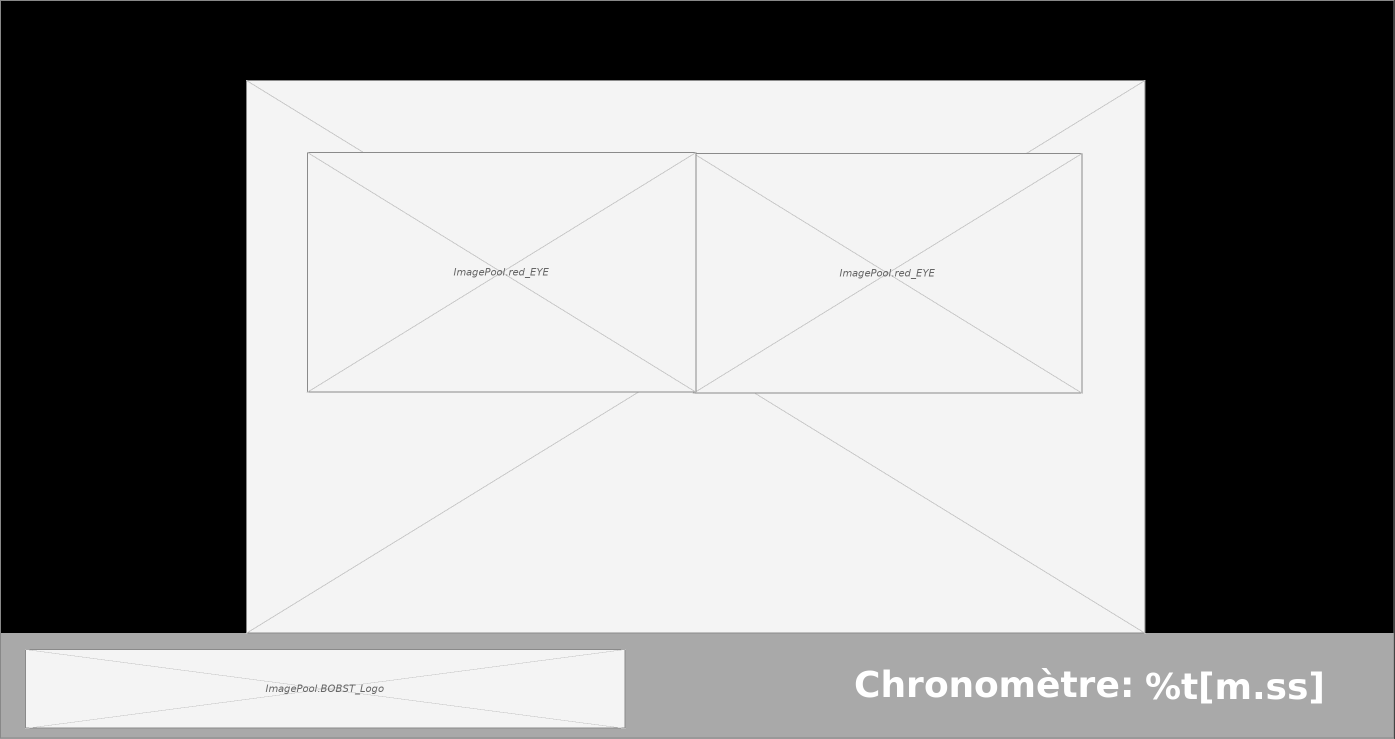
VISUALIZATION V_Match  // 1395x739
    Rectangle (-2,633 1396x109)
    Group (851,647 541x77)
        Label (0,0 400x75), "Chronomètre:"
        Textfield (291,2 250x75), "%t[m.ss]", text variable: G_Match.TimeMatch
    Image (25,649 600x79), image: ImagePool.BOBST_Logo
        OnMouseDown: change screen: V_Menu
    Image (246,80 899x553), image: ImagePool.EYE
    Image (693,153 389x240), invisible if: Not G_Visus.bMatchEnemi, image: ImagePool.red_EYE
    Image (307,152 389x240), invisible if: Not G_Visus.bMatchEnemi, image: ImagePool.red_EYE
END_VISUALIZATION

(* stored: Version 1.1.0.1, ProductVersion 3.1.4024.12
   Visu V_Match: Id {acb41358-2348-4c28-bc62-b6c43509f0cc} *)
